PROGRAM TestProgram

VAR
	bTestVariable : BOOL;
	fTestVariable : REAL;
	nTestVariable : INT;
END_VAR

END_PROGRAM

(* stored: Version 1.1.0.1, ProductVersion 3.1.4024.10
   POU TestProgram: Id {abfc07e4-da28-4e34-a608-54d649b9fe4a}, SpecialFunc None *)
